VAR_GLOBAL
	
	{attribute 'OPC.UA.DA' := '1'}
	{attribute 'OPC.UA.DA.Description' := 'HistoricalAccess with Volatile storage'}
	volatile_sinus	: LREAL;
	{attribute 'OPC.UA.DA' := '1'}
	{attribute 'OPC.UA.DA.Description' := 'HistoricalAccess with Volatile storage'}	
	volatile_cosinus : LREAL;
	{attribute 'OPC.UA.DA' := '1'}
	{attribute 'OPC.UA.DA.Description' := 'HistoricalAccess with Volatile storage'}	
	volatile_cosinushalf : LREAL;
	{attribute 'OPC.UA.DA' := '1'}
	{attribute 'OPC.UA.DA.Description' := 'HistoricalAccess with SQLite storage'}
	sqlite_sinus : LREAL;
	{attribute 'OPC.UA.DA' := '1'}
	{attribute 'OPC.UA.DA.Description' := 'HistoricalAccess with SQLite storage'}	
	sqlite_cosinus : LREAL;
	{attribute 'OPC.UA.DA' := '1'}
	{attribute 'OPC.UA.DA.Description' := 'HistoricalAccess with SQLite storage'}	
	sqlite_cosinushalf : LREAL;

END_VAR

(* stored: Version 1.1.0.1
   GVL GVL_historizing: Id {9dfea3c9-5390-4b35-92a5-198a388c6e05} *)
